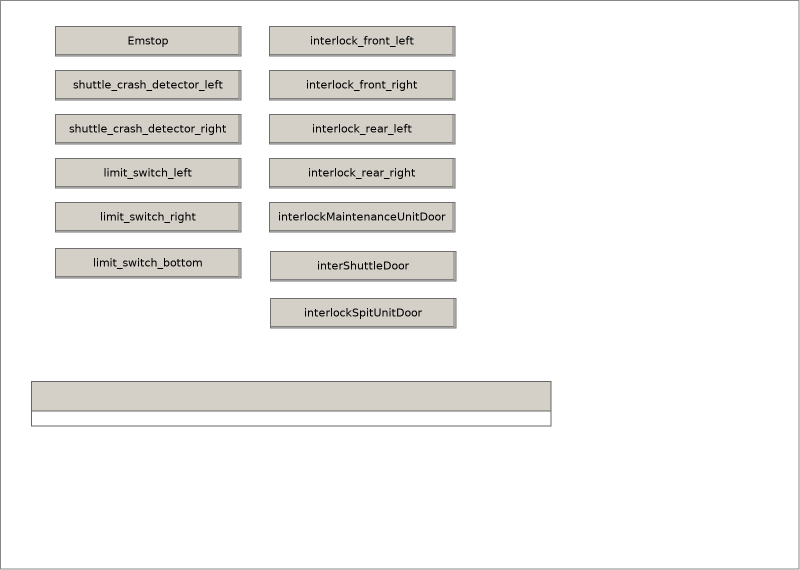
VISUALIZATION VIS_SaftyGuard  // 800x570
    Button (55,26 186x30), "Emstop", colour toggle: GVL_API.stSafetyGuard.emergency_stop
    Button (55,70 186x30), "shuttle_crash_detector_left", colour toggle: GVL_API.stSafetyGuard.shuttle_crash_detector_left
    Button (55,114 186x30), "shuttle_crash_detector_right", colour toggle: GVL_API.stSafetyGuard.shuttle_crash_detector_right
    Button (55,158 186x30), "limit_switch_left", colour toggle: GVL_API.stSafetyGuard.limit_switch_left
    Button (55,202 186x30), "limit_switch_right", colour toggle: GVL_API.stSafetyGuard.limit_switch_right
    Button (269,26 186x30), "interlock_front_left", colour toggle: GVL_API.stSafetyGuard.interlock_front_left
    Button (269,70 186x30), "interlock_front_right", colour toggle: GVL_API.stSafetyGuard.interlock_front_right
    Button (269,114 186x30), "interlock_rear_left", colour toggle: GVL_API.stSafetyGuard.interlock_rear_left
    Button (269,158 186x30), "interlock_rear_right", colour toggle: GVL_API.stSafetyGuard.interlock_rear_right
    Button (269,202 186x30), "interlockMaintenanceUnitDoor", colour toggle: GVL_API.stSafetyGuard.Interlock_maintenace_door, pressed state: P_TwinSAFE.biinterlock[5]
    Button (270,298 186x30), "interlockSpitUnitDoor", colour toggle: GVL_API.stSafetyGuard.Interlock_spit_door
    Button (270,251 186x30), "interShuttleDoor", colour toggle: GVL_API.stSafetyGuard.interlock_shuttle_door
    Button (55,248 186x30), "limit_switch_bottom", colour toggle: GVL_API.stSafetyGuard.limit_switch_bottom
    Table (31,381 520x45), data array: P_SafetyGuard.FB_SafetyGuard
        p3854506369: P_SafetyGuard.FB_SafetyGuard.shuttle_crash_detector
        p1892666644: P_SafetyGuard.FB_SafetyGuard.emergency_stop
        p338671338: P_SafetyGuard.FB_SafetyGuard.limit_switch
        p2170511999: P_SafetyGuard.FB_SafetyGuard.interlock_triggered
        p3723444502: P_SafetyGuard.FB_SafetyGuard.LightCurtainTriggered
        p1218418051: P_SafetyGuard.FB_SafetyGuard.error_code
        p746581629: P_SafetyGuard.FB_SafetyGuard.state
        p3104783080: P_SafetyGuard.FB_SafetyGuard.step
        p2501879983: GVL_API.stSafetyGuard.Initialize
        p7306298: GVL_API.stSafetyGuard.SetOff
        p1037165547: P_SafetyGuard.FB_SafetyGuard.Initialize
        p1488378029: P_SafetyGuard.FB_SafetyGuard.SetOff
        Columns.Column.[5].Template: P_SafetyGuard.FB_SafetyGuard.error_code<>0
        Columns.Column.[8].Template: toggle GVL_API.stSafetyGuard.Initialize
        Columns.Column.[9].Template: toggle GVL_API.stSafetyGuard.SetOff
END_VISUALIZATION

(* stored: Version 1.1.0.1, ProductVersion 3.1.4024.11
   Visu VIS_SaftyGuard: Id {8d8e22a0-6199-4bde-b8a1-9e2a39e3c1ca} *)
